{attribute 'qualified_only'}
VAR_GLOBAL
	sNetId: T_AmsNetId := '5.55.249.199.1.1';
	nPort: T_AmsPort := 851;		
END_VAR

(* stored: Version 1.1.0.1, ProductVersion 3.1.4024.11
   GVL SeparatorAms: Id {3fb81911-5bb4-411a-91d6-940da1f4f474} *)
